FUNCTION TryConvert_UINT_TO_DWORD : BOOL
VAR_INPUT
	in : UINT;
	out : REFERENCE TO DWORD;
END_VAR

out := UINT_TO_DWORD(in);
TryConvert_UINT_TO_DWORD := TRUE;

END_FUNCTION

(* stored: Version 1.1.0.1, ProductVersion 3.1.4024.12
   POU TryConvert_UINT_TO_DWORD: Id {6640dacd-c455-4d76-a33e-49c8f319e780}, SpecialFunc None *)
